FUNCTION_BLOCK EtherCatDeviceWidget
VAR_INPUT
END_VAR
VAR_OUTPUT
END_VAR
VAR
	actualStatus : StatusWidget;
END_VAR
VAR_IN_OUT
	device : EtherCatDevice;
END_VAR

actualStatus(text  := device.actualStatus, 
             color := HealthToColor(device.statuses.healthStatus));

END_FUNCTION_BLOCK

(* stored: Version 1.1.0.1, ProductVersion 3.1.4018.2
   POU EtherCatDeviceWidget: Id {ca672c8c-a49c-4024-9488-7cda63accc71}, SpecialFunc None *)
